PROGRAM MAIN
VAR
END_VAR

JSON_decode();

END_PROGRAM

(* stored: Version 1.1.0.1, ProductVersion 3.1.4024.0
   POU MAIN: Id {1f54d820-f40b-4192-93ef-2e4cd5181e50}, SpecialFunc None *)
